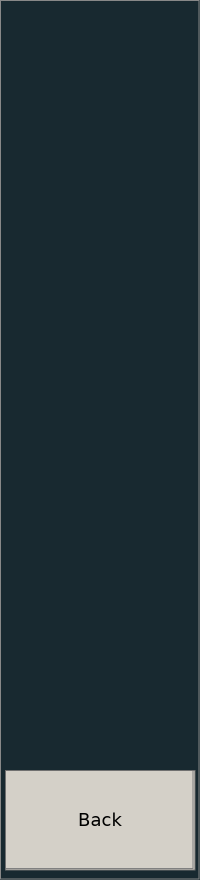
VISUALIZATION NavBarUtilities  // 200x880
VAR_IN_OUT
	btnBack : BOOL;
END_VAR
    Button (5,770 190x100), "Back"
        tap btnBack
END_VISUALIZATION

(* stored: Version 1.1.0.1, ProductVersion 3.1.4024.9
   Visu NavBarUtilities: Id {26047c7b-4ca3-4066-ae53-f9cc15d61b3b} *)
